{attribute 'qualified_only'}
VAR_GLOBAL
	feedback : TxHmi;
	//control : RxHmi;
END_VAR

(* stored: Version 1.1.0.1, ProductVersion 3.1.4020.12
   GVL HMI: Id {852d06cf-bd63-42f7-a1a8-4f24e83802a9} *)
